SUBAPPLICATION Uebung_011b3_PHYSA (* Numeric Value Input ADD with Physical Values *)
  (* Standard: 61499-2; Description: Copyright (c) 2023 Meisterschulen am Ostbahnhof This program and the accompanying materials are made available under the terms of the Eclipse Public License 2.0 which is available at https://www.eclipse.org/legal/epl-2.0/ SPDX-License-Identifier: EPL-2.0 *)
  (* Version 1.0, 2026-04-14, Franz Höpfinger, Meisterschulen am Ostbahnhof, initial API and implementation and/or initial documentation *)
  PACKAGE Uebungen;
  IMPORT Uebungen::const::UT::DefaultPool_Numeric::InputNumber_I3_N;
  IMPORT Uebungen::const::UT::DefaultPool_Numeric::InputNumber_I4_N;
  IMPORT Uebungen::const::UT::DefaultPool_Numeric::OutputNumber_N3_N;
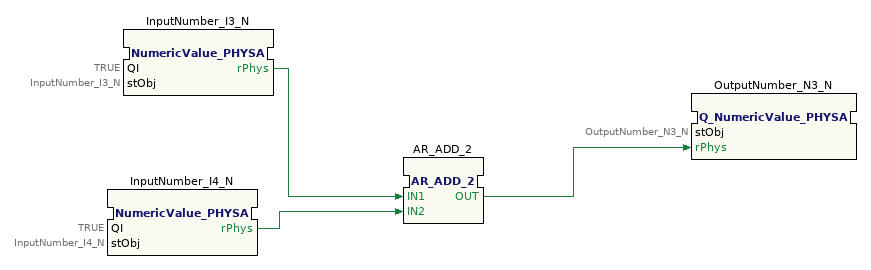
  FBS
    InputNumber_I3_N : isobus::UT::io::NumericValue::NumericValue_PHYSA(QI := TRUE, stObj := InputNumber_I3_N);
    InputNumber_I4_N : isobus::UT::io::NumericValue::NumericValue_PHYSA(QI := TRUE, stObj := InputNumber_I4_N);
    AR_ADD_2 : adapter::iec61131::arithmetic::AR_ADD_2;
    OutputNumber_N3_N : isobus::UT::Q::Q_NumericValue_PHYSA(stObj := OutputNumber_N3_N);
  END_FBS
  ADAPTER_CONNECTIONS
    InputNumber_I3_N.rPhys TO AR_ADD_2.IN1;
    InputNumber_I4_N.rPhys TO AR_ADD_2.IN2;
    AR_ADD_2.OUT TO OutputNumber_N3_N.rPhys;
  END_CONNECTIONS
END_SUBAPPLICATION
